// TIA Portal project "Lab_3_Funksjonsblokk" (V15.1)

(* hardware
DEVICE "ET 200SP station_1"  ET 200SP-Station
   slot 0: "Rack_0"  Rack  6ES5 710-8MAx1
   slot 1: "PLC_1"  CPU 1512SP F-1 PN  6ES7 512-1SK01-0AB0  V2.6
   slot 2: "DI 8x24VDC HF_1"  DI 8x24VDC HF  6ES7 131-6BF00-0CA0  V2.0
      slot 1: "DI 8x24VDC HF_1"  DI 8x24VDC HF
   slot 3: "DI 8x24VDC HF_2"  DI 8x24VDC HF  6ES7 131-6BF00-0CA0  V2.0
      slot 1: "DI 8x24VDC HF_2"  DI 8x24VDC HF
   slot 4: "DQ 8x24VDC/0.5A HF_1"  DQ 8x24VDC/0.5A HF  6ES7 132-6BF00-0CA0  V2.0
      slot 1: "DQ 8x24VDC/0.5A HF_1"  DQ 8x24VDC/0.5A HF
   slot 5: "DQ 8x24VDC/0.5A HF_2"  DQ 8x24VDC/0.5A HF  6ES7 132-6BF00-0CA0  V2.0
      slot 1: "DQ 8x24VDC/0.5A HF_2"  DQ 8x24VDC/0.5A HF
   slot 6: "CM 4xIO-Link_1"  CM 4xIO-Link  6ES7 137-6BD00-0BA0  V2.2
      slot 1: "CM 4xIO-Link_1"  6ES7 137-6BD00-0BA0
   slot 7: "Server module_1"  Server module  6ES7 193-6PA00-0AA0  V1.1
      slot 1: "Server module_1"  Server module
   slot 127: "BA 2xRJ45"  BA 2xRJ45  6ES7 193-6AR00-0AA0  V0.0
      slot 32769: "Port_1"  6ES7 193-6AR00-0AA0
      slot 32770: "Port_2"  6ES7 193-6AR00-0AA0
*)

// ===== PLC "PLC_1"  CPU 1512SP F-1 PN =====

VAR_GLOBAL   // PLC tag table "gtIDrilling"
   "start_btn" AT %I1.0 : Bool;   // True = Start button pushed
   "stop_btn" AT %I1.1 : Bool;   // False = Stop button pushed
   "op-mode_btn" AT %I1.2 : Bool;   // Select operation mode (False = Setup mode, True = Automatic mode)
   "reset_btn" AT %I1.3 : Bool;   // True = Reset button pushed
   "carrier_stopper_pos" AT %I1.4 : Bool;   // True = Carrier detected at stopper position (corresponds to ident code bit 0)
   "emergency_stop_btn" AT %I1.5 : Bool;   // False = Emergency stop button pushed (n.c.)
   "carrier_entry_pos" AT %I1.6 : Bool;   // True = Carrier detected at conveyor entry
   "carrier_exit_pos" AT %I1.7 : Bool;   // True = Carrier detected at conveyor exit
   "carrier_ident_0" AT %I42.0 : Bool;   // True = Carrier ident code bit 0 detected
   "carrier_ident_1" AT %I42.1 : Bool;   // True = Carrier ident code bit 1 detected
   "carrier_ident_2" AT %I42.2 : Bool;   // True = Carrier ident code bit 2 detected
   "carrier_ident_3" AT %I42.3 : Bool;   // True = Carrier ident code bit 3 detected
   "switch_S1" AT %I42.4 : Bool;   // A = True = Encoder A signal detcted, R = False = Coupling signal right detected
   "switch_S2" AT %I42.5 : Bool;   // B = True = Encoder B signal detected, L = False = Coupling signal left detected
   "stop_cylinder_low_pos" AT %I42.7 : Bool;   // True = Stopper cylinder in lower end position
   "start_btn_light" AT %Q1.0 : Bool;   // True = Switch on start button signal light
   "reset_btn_light" AT %Q1.1 : Bool;   // True = Switch on reset button signal light
   "func_Q1_light" AT %Q1.2 : Bool;   // True = Switch on special function Q1 signal light
   "func_Q2_light" AT %Q1.3 : Bool;   // True = Switch on special function Q2 signal light
   "belt_forward" AT %Q1.4 : Bool;   // True = Drive belt in forward direction
   "belt_reverse" AT %Q1.5 : Bool;   // True = Drive belt in reverse direction
   "belt_speed" AT %Q1.6 : Bool;   // Select belt speed (False = normal, True = slow)
   "move_cylinder_down" AT %Q1.7 : Bool;   // True = Move stopper cylinder down
   "coupling_signal_left" AT %Q42.4 : Bool;   // True = Send coupling signal left
   "coupling_signal_right" AT %Q42.5 : Bool;   // True = Send coupling signal right
   "X-axix_left_end_pos" AT %I0.0 : Bool;   // True = drill in X-axis left posistion
   "X-axis_right_pos" AT %I0.1 : Bool;   // True = drill in X-axis right posistion
   "front_cover_correct" AT %I0.2 : Bool;   // True = front cover correct after inspection
   "front_cover_present" AT %I0.3 : Bool;   // True = front cover present
   "Z-axis_upper_pos" AT %I0.4 : Bool;   // True = drill in Z-axis upper posistion
   "Z_axis_lower_pos" AT %I0.5 : Bool;   // True = drill in Z-axis lower posistion
   "back_cover_present" AT %I0.7 : Bool;   // True = Back cover present on workpiece
   "move_X-axis_left" AT %Q0.0 : Bool;   // True = drill will move to X-axis left posistion
   "move_X-axis_right" AT %Q0.1 : Bool;   // True = drill will move to X-axis right posistion
   "switch_drill_1" AT %Q0.2 : Bool;   // True = drill 1 will start drilling
   "switch_drill_2" AT %Q0.3 : Bool;   // True = drill 2 will start drilling
   "move_Z-axis_up" AT %Q0.4 : Bool;   // True = drill will move to Z-axis upper posistion
   "move_Z-axis_down" AT %Q0.5 : Bool;   // True = drill will move to Z-axis lower posistion
   "open_Z-axis_end_pos_lock" AT %Q0.6 : Bool;   // True = drill is allowed to move up or down
END_VAR

DATA_BLOCK "fbIDrilling_DB"   // DB1
{ S7_Optimized_Access := 'TRUE' }
VERSION : 0.1
// stored: InstanceOfName fbIDrilling
"fbIDrilling"
BEGIN
END_DATA_BLOCK

// folder: System blocks/Program resources

DATA_BLOCK "Timer"   // DB2
{ S7_Optimized_Access := 'TRUE' }
AUTHOR : Simatic
FAMILY : IEC
NAME : IEC_TMR
VERSION : 1.0
// stored: InstanceOfName IEC_TIMER
"IEC_TIMER"
BEGIN
END_DATA_BLOCK

// folder: (top level)

FUNCTION_BLOCK "fbIDrilling"   // FB1, SCL
{ S7_Optimized_Access := 'TRUE' }
VERSION : 0.1
   VAR_INPUT
      Xstartbtn : Bool;
      Xstoppbtn : Bool;
      Xreset_btn : Bool;
      Xcarrier_stopper_pos : Bool;
      Xcarrier_entry_pos : Bool;
      Xcarrier_exit_pos : Bool;
      "XX-axis_left" : Bool;
      "XX-axis_right" : Bool;
      "XZ-axis_up" : Bool;
      "XZ-axis_down" : Bool;
      Xop_mode_switch : Bool;
      Xback_cover_present : Bool;
   END_VAR
   VAR_OUTPUT
      Ystart_btn_light : Bool;
      Ybelt_forward : Bool;
      Yreset_btn : Bool;
      Ymove_X_axis_left : Bool;
      Ymove_X_axis_right : Bool;
      Ydrill_1_on : Bool;
      Ydrill_2_on : Bool;
      Ymove_Z_axis_down : Bool;
      Ymove_Z_axis_up : Bool;
      Yopen_Z_axis_lock : Bool;
      Ymove_cylinder_down : Bool;
   END_VAR
   VAR
      stTimeNow : Time;
      sbTimerFinnished : Bool;
   END_VAR
BEGIN
   (*
   ---------------------------------------------------------------------------------------------------------
   Conveyer belt:
   *)

   //Get's the conveyer to drive in automatic mode
   IF #Xop_mode_switch = TRUE THEN                       //When true, initialize automatic mode
       IF #Xcarrier_entry_pos = TRUE THEN                //Checks if workpiece is present on belt
           #Ybelt_forward := TRUE;                       //Starts moving the belt
       END_IF;
       IF #Xcarrier_exit_pos = TRUE THEN                 //If the workpiece is at the end of the belt
           #Ybelt_forward := FALSE;                      //Stops the belt from moving
       END_IF;
   ELSE                                                  //If the switch is in manual mode
       IF #Xstartbtn = TRUE THEN                         //If the start button is pressed
           #Ystart_btn_light := TRUE;                    //Starts the start button light
           #Ybelt_forward    := TRUE;                    //Starts the belt moving forward
       END_IF;
       IF #Xstoppbtn = FALSE THEN                        //If the stop button is pressed
           #Ystart_btn_light := FALSE;                   //Turns off the start button light
           #Ybelt_forward    := FALSE;                   //Stops the belt moving
       END_IF;
   END_IF;

   //Timer to stop the workpiece at the middle of the belt
   "Timer".TON(IN:=#Xcarrier_stopper_pos,                 //Checks if workpiece is in middle of belt
               PT:=T#5s,                                  //Stops for 5 sekunds
               Q=>#sbTimerFinnished,                         //Boolean output for timer, true when finnished
               ET=>#stTimeNow);                            //Static timer to show time during timing


   (*
   -----------------------------------------------------------------------------------------------------------
   iDrilling modul:
   *)

   //Resets timer when not triggered
   IF NOT #Xcarrier_stopper_pos THEN                       //Checks if there is not a workpiece in the middle of the belt
       RESET_TIMER("Timer");                               //Resets the timer
       #Ymove_cylinder_down := FALSE;                      //Moves the cylinder down, so it ready for the next
   ;
   END_IF;

   //Puts the drill back at it's initial posistion
   #Yopen_Z_axis_lock  := TRUE;                             //Opens the lock, so the drill can move in Z-direction
   #Ymove_Z_axis_up    := TRUE;                             //Moves the drill up in Z-direction
   #Ymove_Z_axis_down  := FALSE;                            //This is false so the two outputs don't contradicts eachother
   #Ymove_X_axis_right := TRUE;                             //Moves the drill to right in X-direction
   #Ymove_X_axis_left  := FALSE;                            //Turns the X-axis left to false so it dosen't contradict the right command
   #Ydrill_1_on        := FALSE;                            //Turns drill1 off
   #Ydrill_2_on        := FALSE;                            //Turns drill2 off
   //#Yopen_Z_axis_lock  := FALSE;                          //Closes the lock again

   //Drills the workpiece for the set time in "Timer" ("Timer".PT)
   IF (NOT #sbTimerFinnished) AND #Xcarrier_stopper_pos AND #Xback_cover_present THEN   //If the timer is not finnished, and there is a workpiece at the middle of the belt
       #Ydrill_1_on        := TRUE;                         //Turns drill1 on
       #Ydrill_2_on        := TRUE;                         //Turns drill2 on
       #Yopen_Z_axis_lock  := TRUE;                         //Opens the lock, so the drill can move in Z-direction
       #Ymove_X_axis_right := TRUE;                         //Moves the drill to right in the X-axis
       #Ymove_X_axis_left  := FALSE;                        //Turns the X-axis left to false so it dosen't contradict the right command
       #Ymove_Z_axis_up    := FALSE;                        //Turns the Z-axis up to false so it dosen't contradict the down command
       #Ymove_Z_axis_down  := TRUE;                         //Puts the drill down in Z-axis, so it can start drilling
   ;
   END_IF;

   //Sends the workpiece forward after it's been drilled
   IF #sbTimerFinnished AND #Xcarrier_stopper_pos THEN      //If the timer is finnished and the workpiece is still at the middle of the belt
      #Ymove_cylinder_down  := TRUE;                        //Moves the cylinder down, so the belt can send it forward
   ;
   END_IF;

   IF #Xcarrier_stopper_pos AND (NOT #Xback_cover_present) THEN    //If the back cover is not present, we cannot drill
       #Ymove_cylinder_down  := TRUE;                        //So we send it forward
   ;
   END_IF;
END_FUNCTION_BLOCK

FUNCTION_BLOCK "Block_1"   // FB2, FBD
{ S7_Optimized_Access := 'TRUE' }
VERSION : 0.1
BEGIN
END_FUNCTION_BLOCK

ORGANIZATION_BLOCK "Main"   // OB1, FBD, ProgramCycle
TITLE = "Main Program Sweep (Cycle)"
{ S7_Optimized_Access := 'TRUE' }
VERSION : 0.1
   VAR_INPUT
      Initial_Call : Bool;   // Initial call of this OB
      Remanence : Bool;   // =True, if remanent data are available
   END_VAR
BEGIN

REGION Network 1
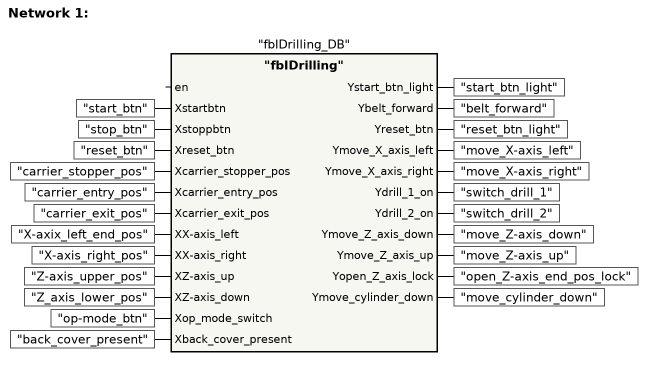
   "fbIDrilling_DB"(Xstartbtn := "start_btn",   // "fbIDrilling"
                    Xstoppbtn := "stop_btn",
                    Xreset_btn := "reset_btn",
                    Xcarrier_stopper_pos := "carrier_stopper_pos",
                    Xcarrier_entry_pos := "carrier_entry_pos",
                    Xcarrier_exit_pos := "carrier_exit_pos",
                    "XX-axis_left" := "X-axix_left_end_pos",
                    "XX-axis_right" := "X-axis_right_pos",
                    "XZ-axis_up" := "Z-axis_upper_pos",
                    "XZ-axis_down" := "Z_axis_lower_pos",
                    Xop_mode_switch := "op-mode_btn",
                    Xback_cover_present := "back_cover_present",
                    Ystart_btn_light => "start_btn_light",
                    Ybelt_forward => "belt_forward",
                    Yreset_btn => "reset_btn_light",
                    Ymove_X_axis_left => "move_X-axis_left",
                    Ymove_X_axis_right => "move_X-axis_right",
                    Ydrill_1_on => "switch_drill_1",
                    Ydrill_2_on => "switch_drill_2",
                    Ymove_Z_axis_down => "move_Z-axis_down",
                    Ymove_Z_axis_up => "move_Z-axis_up",
                    Yopen_Z_axis_lock => "open_Z-axis_end_pos_lock",
                    Ymove_cylinder_down => "move_cylinder_down");
END_REGION
END_ORGANIZATION_BLOCK